FUNCTION_BLOCK IntToBool (* Basic Function Block Type *)
  (* Standard: 61499-2 *)
  (* Version 0.0, 11/21/2016, chivdan, nxtControl GmbH, Template *)
  PACKAGE Main;
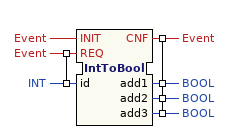
  EVENT_INPUT
    INIT;
    REQ WITH id; (* Normal Execution Request *)
  END_EVENT
  EVENT_OUTPUT
    CNF WITH add1, add2, add3; (* Execution Confirmation *)
  END_EVENT
  VAR_INPUT
    id : INT; (* Input event qualifier *)
  END_VAR
  VAR_OUTPUT
    add1 : BOOL;
    add2 : BOOL;
    add3 : BOOL;
  END_VAR
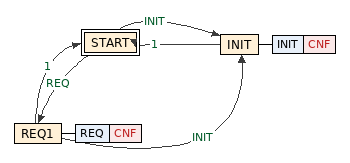
  EC_STATES
    START; (* Initial State *)
    REQ1 : REQ -> CNF; (* Normal execution *)
    INIT : INIT -> CNF;
  END_STATES
  EC_TRANSITIONS
    START TO REQ1 := REQ;
    REQ1 TO START := 1;
    START TO INIT := INIT;
    INIT TO START := 1;
    REQ1 TO INIT := INIT;
  END_TRANSITIONS
  ALGORITHM INIT IN ST: (* Initialization algorithm *)
add1:=FALSE;
add2:=FALSE;
add3:=FALSE;
  END_ALGORITHM
  ALGORITHM REQ IN ST: (* Normally executed algorithm *)
;
IF id = 1 THEN
	add1:=TRUE;
	add2:=FALSE;
	add3:=FALSE;
ELSIF id = 2 THEN
	add1:=FALSE;
	add2:=TRUE;
	add3:=FALSE;
ELSIF id = 3 THEN
	add1:=FALSE;
	add2:=FALSE;
	add3:=TRUE;
ELSE
	add1:=FALSE;
	add2:=FALSE;
	add3:=FALSE;
END_IF;
  END_ALGORITHM
END_FUNCTION_BLOCK
